# EPICS autosave request: iocs/vimbaIOC/iocBoot/iocVimba/auto_settings.req
file "ADVimba_settings.req",              P=$(P),  R=cam1:
file "NDStdArrays_settings.req",          P=$(P),  R=image1:
file "commonPlugin_settings.req",         P=$(P)
